Fanuc KAREL source: ko00098.KL

-- PROVISIONAL review KL for V770-1; original PC SHA256 4036c813a6c17a44e4931d8736cc79444c13447eee4fd6fa75985e1fe871668f
-- Incomplete behavior may be omitted. Consult companion uncertainty JSON. Do not deploy.
PROGRAM KO00098
%NOLOCKGROUP
VAR
  A : INTEGER
  B : INTEGER
  OUT : REAL
BEGIN
  -- UNRESOLVED_PC offsets 5-12; opcodes 9D,23
  -- UNRESOLVED_PC offsets 17-28; opcodes 2E,23
  -- UNRESOLVED_PC offsets 33-58; opcodes 27,27,21,64,27,21,64,76,23
  -- UNRESOLVED_PC offsets 63-67; opcodes 7F
END KO00098
